PROGRAM VltE2E_splice_stable
VAR
	a : BOOL;
	b : BOOL;
	out1 : BOOL;
	out2 : BOOL;
END_VAR

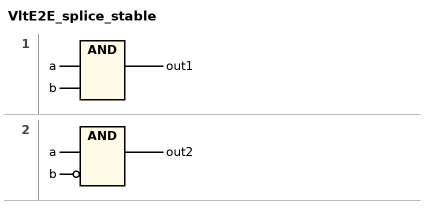
// NETWORK 1
out1 := a AND b;

// NETWORK 2
out2 := a AND NOT b;

END_PROGRAM

(* stored: Version 1.1.0.1, ProductVersion 3.1.4024.16
   POU VltE2E_splice_stable: Id {7ff752c2-5c75-4434-a49e-6a4d4def900b}, SpecialFunc None *)
